Fanuc KAREL source: ka00089.KL

-- PROVISIONAL review KL for V1013-1; original PC SHA256 cef9d7c927dca21828e53fe39bce2ac82943881c434f1cfa0da68c408dbc17fe
-- Incomplete behavior may be omitted. Consult companion uncertainty JSON. Do not deploy.
PROGRAM KA00089
%NOLOCKGROUP
-- UNRESOLVED_DECL SRC type=000199
-- UNRESOLVED_DECL DST type=000101
BEGIN
  -- UNRESOLVED_PC offsets 5-25; opcodes 49,7E,4A
  -- UNRESOLVED_PC offsets 30-34; opcodes 7F
END KA00089
